(*********************************** G.D S.p.A. - Technical Department ***********************************
============= PROGRAM INFO ============
FOLDER:             TBD
MACHINES INVOLVED:  TBD 

============= DESCRIPTION =============

============= REVISIONS ===============
Date		Version	 	Author      	Description             
----------	-------		------------  	--------------------------------------------
2019/04/24 	0000.00	 	M.Grasso		Creation of the PRG

**********************************************************************************************************)
(*$R 
	process_ref:= prc; 
$*)
PROGRAM csp_transfer_main_safety_drives_SD41100
VAR
	prc:					process;
	prc_path:				STRING;	

	sig:					safety_integrated_group;
	chA_smes_sis:			safety_integrated_series;
	chB_smes_sis:			safety_integrated_series;
END_VAR

_read_var_input();

_objects_manager();

IF NOT objects_running()
THEN
	RETURN;	
END_IF

_read_process_image();

_mode_manager();

safety_integrated_series_close(chA_smes_sis);
safety_integrated_series_close(chB_smes_sis);

CASE process_get_mode(prc) OF
	MODE_ABSENT,
	MODE_INACTIVE:
		RETURN;
	MODE_TEST:
		;
END_CASE

_set_runtime_properties();

(********************************* BODY *********************************)

(************************************************************************)

_handle_messages();

_write_output();

ACTION _handle_messages:
;
END_ACTION

ACTION _handle_process_test:
;
END_ACTION

ACTION _mode_manager:
IF process_mode_req_is_pending(prc)
THEN
    process_apply_mode_req_first_step(prc);
    CASE process_get_mode(prc) OF
        MODE_TO_ABSENT:
			;
        MODE_TO_INACTIVE:
			;
        MODE_TO_TEST:
			;
        MODE_TO_OPERATIONAL:
			;
    END_CASE
    process_apply_mode_req_second_step(prc);
END_IF
END_ACTION

ACTION _objects_manager:
IF objects_initialization()
THEN
	sub_process_init(
		object_name					:= 'csp_transfer_main_safety_drives.prc', 
		process						:= csp_transfer_main_safety.prc, 
		CONVERSION_this				:= prc);
		
	prc_path 						:= process_get_path(prc);

	safety_integrated_group_init(
        object_name				:=	CONCAT(prc_path, '_sig'), 
		controller				:=	csp_transfer_main_safety_interface.SPLC40210_sic,
        process					:=	prc,
        CONVERSION_this			:=	sig);

	(* Channel A SMES series *)
	safety_integrated_series_init(
		object_name				:=	CONCAT(prc_path, '_chA_smes_sis'), 
		_type					:=	SAFETY_INTEGRATED_SERIES_TYPE_NO_RESET,
		discrepancy_active		:=	TRUE,
		forced_open_active		:=	TRUE,
		process					:=	prc,
		CONVERSION_this			:=	chA_smes_sis);

	safety_integrated_series_add_safety_integrated_group(
		group					:=	sig,
		CONVERSION_this			:=	chA_smes_sis);

	safety_integrated_series_add_safety_integrated_series(
		series_active			:=	TRUE,
		series_polarity_direct	:=	TRUE,
		contact					:=	csp_transfer_main_safety_drives_commonConfiguration.rack_smes_sis, (*Marco : To be checked*)
		CONVERSION_this			:=	chA_smes_sis);
		
	(* Channel B SMES series *)
	safety_integrated_series_init(
		object_name				:=	CONCAT(prc_path, '_chB_smes_sis'), 
		_type					:=	SAFETY_INTEGRATED_SERIES_TYPE_NO_RESET,
		discrepancy_active		:=	TRUE,
		forced_open_active		:=	TRUE,
		process					:=	prc,
		CONVERSION_this			:=	chB_smes_sis);

	safety_integrated_series_add_safety_integrated_group(
		group					:=	sig,
		CONVERSION_this			:=	chB_smes_sis);
		
	safety_integrated_series_add_safety_integrated_series(
		series_active			:=	TRUE,
		series_polarity_direct	:=	TRUE,
		contact					:=	csp_transfer_main_safety_drives_commonConfiguration.rack_smes_sis, (*Marco : To be checked*)
		CONVERSION_this			:=	chB_smes_sis);
		
END_IF

IF objects_running()
THEN
	process_cycle(prc);
  	safety_integrated_group_cycle(sig);
	safety_integrated_series_cycle(chA_smes_sis);
	safety_integrated_series_cycle(chB_smes_sis);
END_IF
END_ACTION

ACTION _read_process_image:
;
END_ACTION

ACTION _read_var_input:
;
END_ACTION

ACTION _set_runtime_properties:
;
END_ACTION

ACTION _write_output:
;
END_ACTION

END_PROGRAM

(* stored: Version 1.1.0.1, ProductVersion 3.1.4024.3
   POU csp_transfer_main_safety_drives_SD41100: Id {a6ac0313-05a7-40e4-a29c-b428f2214b40}, SpecialFunc None
   Action _handle_messages: Id {e864c5cb-c6ad-4838-96ee-3e7902f5a877}
   Action _handle_process_test: Id {5049892c-8817-4e1e-82bd-d0af5f9818dd}
   Action _mode_manager: Id {f90156c5-be4c-4ebf-aab9-1bbe71f73fb6}
   Action _objects_manager: Id {803e7d72-afb7-4786-83ed-c2aa86c7d1cf}
   Action _read_process_image: Id {8e7cf120-b72f-45dc-9b7c-0b8e903694a5}
   Action _read_var_input: Id {d324da39-5801-494b-a56f-6e779fd29f02}
   Action _set_runtime_properties: Id {f4f49bd6-f49b-468a-acef-f202b1bac4ae}
   Action _write_output: Id {c37e9ceb-abcc-40e2-842a-f3751927f118} *)
